FUNCTION_BLOCK FB_Logik_ShortestDistance IMPLEMENTS ITF_Fahrlogik
VAR_INPUT
END_VAR
VAR_OUTPUT
END_VAR
VAR
END_VAR

{warning 'Methodenimplementierung hinzufügen'}
METHOD M_getNextTask : ST_Fahrauftrag
VAR_INPUT
	LiftStockwerkAktuell	: INT;
END_VAR
VAR_IN_OUT
	(* Die Liste zum Durchsuchen*)
	Auftraege	: ARRAY [1..10] OF ST_Fahrauftrag;
END_VAR
VAR
	i : DINT;
    BestIndex : DINT := 0;
    shortestDistance  : INT := 100; // Startwert extrem hoch setzen
    Distance     : INT;
    Leer       : ST_Fahrauftrag;
END_VAR

FOR i := 1 TO UPPER_BOUND(Auftraege, 1) DO
	
IF Auftraege[i].istAktiv THEN
	Distance := ABS(Auftraege[i].Startstockwerk - Divers.AktuellesStockwerk);
	
	IF Distance < shortestDistance THEN
		shortestDistance := Distance;
		BestIndex := i;
	END_IF
END_IF
END_FOR

IF BestIndex > 0 THEN
	M_getNextTask := Auftraege[BestIndex];
ELSE
	M_getNextTask := Leer;
END_IF
END_METHOD

END_FUNCTION_BLOCK

(* stored: Version 1.1.0.1
   POU FB_Logik_ShortestDistance: Id {fab64295-45fd-49b6-9a64-446951ceeeb8}, SpecialFunc None
   Method M_getNextTask: Id {31eb2968-912d-4f8c-825d-e5018b0d2b16} *)
